{attribute 'GeneratedUsingTerminal: EP2316-0008-0016'}
{attribute addProperty BoxType "EP2316-0008-0016"}
{attribute addProperty Id "Diag_InputAT %I*ARRAY[0..7] OF BOOL8"}
{attribute addProperty CRC "568896300"}
{attribute addProperty Size "8"}
TYPE DO_Diag_Inputs_584303BF EXTENDS InputBase_8311D824 :
STRUCT
	{attribute addProperty Name "Diag_Input"}
	Diag_Input AT %I* : ARRAY[0..7] OF BOOL;
END_STRUCT
END_TYPE

(* stored: Version 1.2.0.0, ProductVersion 3.1.4024.9
   DUT DO_Diag_Inputs_584303BF: Id {459c0b67-c9d8-4bc1-924a-9e1781e15741} *)
